Yaskawa INFORM job: R1_W18,19,21(0,0)_KM-OKNEW_MP.JBI

/JOB
//NAME R1_W18,19,21(0,0)_KM-OKNEW_MP
///FOLDERNAME SCIANA-NOWY-R2-KM
//POS
///NPOS 80,80,0,5,0,0
///TOOL 0
///POSTYPE PULSE
///PULSE
C00000=160147,-53341,-73853,12461,99147,-87592
C00001=218993,-28852,-38707,63009,50059,-50724
C00002=220406,-26361,-36985,62252,49273,-50314
C00003=220646,-24565,-35727,62034,49192,-50185
C00004=230254,-40887,-46835,45385,32404,-42165
C00005=230400,-39401,-45908,45036,32465,-41986
C00006=231234,-39623,-46051,44273,32027,-41630
C00007=229297,-43449,-48422,46653,32652,-42787
C00008=220299,-31016,-30594,80800,44642,-56707
C00009=217027,-34239,-32011,82093,46850,-57475
C00010=218993,-28852,-38707,63009,50059,-50724
C00011=218994,-27956,-30243,66729,47934,-53296
C00012=220309,-26407,-29170,66164,47121,-52969
C00013=220627,-24126,-27569,65891,46994,-52801
C00014=226141,-36155,-35714,59251,35589,-49390
C00015=226354,-34126,-34390,58846,35579,-49175
C00016=227436,-34522,-34649,58234,34891,-48867
C00017=226354,-34126,-34390,58846,35579,-49175
C00018=223002,-47340,-42625,62762,36811,-51283
C00019=212788,-54368,-45816,77108,46096,-57028
C00020=192935,-54093,-45665,79683,60227,-58916
C00021=199706,-75247,-47809,90044,85458,-59697
C00022=-183741,-84985,-51911,-73844,36583,24995
C00023=-167288,13673,-10685,-75581,87166,55635
C00024=-170115,12447,-11796,-75038,85255,55349
C00025=-171924,12238,-11987,-74680,84031,55173
C00026=-172522,13420,-10920,-74565,83613,55136
C00027=-171924,12238,-11987,-74680,84031,55173
C00028=-174289,-8390,-27193,-73022,70502,53860
C00029=-175043,-10382,-28758,-72859,69972,53803
C00030=-173781,-9335,-27936,-73156,70837,53929
C00031=-170061,7965,-6237,-85273,82617,57097
C00032=-170115,12447,-11796,-75038,85255,55349
C00033=-170854,10317,-178,-75577,82417,58957
C00034=-171936,11268,672,-75477,81652,58870
C00035=-172588,12571,1843,-75403,81184,58831
C00036=-173506,-7047,-14827,-73481,70592,57186
C00037=-174065,-6013,-13997,-73389,70213,57115
C00038=-174718,-7755,-15385,-73301,69749,57060
C00039=-174065,-6013,-13997,-73389,70213,57115
C00040=-167494,-6216,-14159,-74323,74762,57821
C00041=-167212,9242,-4388,-85630,84611,57426
C00042=-171443,11016,-20134,-69762,86873,53798
C00043=-159366,28260,10505,-84577,79142,62797
C00044=-161376,29134,12959,-84526,77561,63200
C00045=-170734,9630,-20866,-69941,87234,53997
C00046=-170910,12626,-18186,-69900,87078,54023
C00047=-161329,41068,52798,-88533,75848,71873
C00048=-156885,52620,73245,-89064,78615,75095
C00049=-156885,42414,52033,-87693,79106,71429
C00050=-156885,42414,52033,-87693,79106,71429
C00051=-170734,9630,-20866,-69941,87234,53997
C00052=-170910,12626,-18186,-69900,87078,54023
C00053=-157101,42923,53642,-87848,78897,71764
C00054=-152830,31819,8463,-85121,84190,61637
C00055=-158696,27639,4326,-84119,80078,61206
C00056=-161292,29017,11142,-84335,77760,62716
C00057=-170734,9630,-20866,-69941,87234,53997
C00058=-170910,12626,-18186,-69900,87078,54023
C00059=-161298,39658,49489,-88232,75954,71262
C00060=-157285,44272,54296,-87830,78791,71632
C00061=-149677,12279,17067,-86345,84838,68845
C00062=-232880,-71521,-75686,35941,36210,-39067
C00063=-222816,-51916,-50111,20966,8363,-34041
C00064=-221849,-36521,-38911,13718,8860,-30841
C00065=-232908,-27541,-49501,31528,41666,-36518
C00066=-231674,-29527,-50857,30509,41069,-36068
C00067=-221749,-36952,-39190,13316,8793,-30662
C00068=-222742,-43680,-43403,19802,8163,-33549
C00069=-222742,-43680,-43403,19802,8163,-33549
C00070=-222596,-43007,-42997,18855,8220,-33127
C00071=-222188,-38344,-40086,15669,8713,-31707
C00072=-221923,-38189,-39826,14529,8586,-31201
C00073=-222612,-48256,-49120,16792,9247,-32198
C00074=-222612,-48582,-51707,14592,10621,-31204
C00075=-222673,-45322,-48482,15253,10333,-31500
C00076=-222605,-45676,-48694,15053,10272,-31413
C00077=-229461,-68293,-61058,53300,9643,-48481
C00078=-91363,-148629,-70156,-110021,65590,32869
C00079=-795,-65919,-41644,-5435,89623,77465
BC00000=340583,1203205,1070892
BC00001=395849,1203429,1070910
BC00002=395849,1203429,1070910
BC00003=395849,1203429,1070910
BC00004=395849,1203429,1070910
BC00005=395849,1203429,1070910
BC00006=395849,1203429,1070910
BC00007=395849,1203429,1070910
BC00008=395849,1203429,1070910
BC00009=395849,1203429,1070910
BC00010=395849,1203429,1070910
BC00011=395849,1203429,690394
BC00012=395849,1203429,690394
BC00013=395849,1203429,690394
BC00014=395849,1203429,690394
BC00015=395849,1203429,690394
BC00016=395849,1203429,690394
BC00017=395849,1203429,690394
BC00018=395849,1203429,690394
BC00019=395849,1203429,886238
BC00020=395849,1203429,886238
BC00021=392558,1157770,1067511
BC00022=392558,972054,1067511
BC00023=363587,801900,1037584
BC00024=363587,805740,1037584
BC00025=363587,805740,1037584
BC00026=363587,805740,1037584
BC00027=363587,805740,1037584
BC00028=363587,805740,1037584
BC00029=363587,805740,1037584
BC00030=363587,805740,1037584
BC00031=363587,805740,1037584
BC00032=363587,805740,1037584
BC00033=363587,805740,689443
BC00034=363587,805740,689443
BC00035=363586,805740,689440
BC00036=363587,805740,689443
BC00037=363587,805740,689443
BC00038=363587,805740,689443
BC00039=363587,805740,689443
BC00040=363587,805740,689443
BC00041=363587,805740,1037584
BC00042=366059,811819,1070910
BC00043=358283,754245,1070910
BC00044=358283,754245,1070910
BC00045=358283,754245,1070910
BC00046=358283,754245,1070910
BC00047=358283,754245,1070910
BC00048=358283,754245,1069404
BC00049=352744,750822,887513
BC00050=348457,746222,883985
BC00051=358283,754245,1070910
BC00052=358283,754245,1070910
BC00053=348457,746222,705777
BC00054=358284,754245,886289
BC00055=358284,754245,886289
BC00056=358283,754245,886291
BC00057=358283,754245,1070910
BC00058=358283,754245,1070910
BC00059=358283,754245,886291
BC00060=358283,754245,885920
BC00061=358283,794942,867656
BC00062=395849,1135044,1070910
BC00063=395849,1140911,1070910
BC00064=395849,1140998,1070910
BC00065=395849,1142547,1070910
BC00066=395849,1142547,1070910
BC00067=395849,1140998,895189
BC00068=395849,1140998,895189
BC00069=395849,1140998,721535
BC00070=394321,1142791,721535
BC00071=394321,1142791,721535
BC00072=394321,1142791,532615
BC00073=394321,1142791,532615
BC00074=394321,1142791,868876
BC00075=387636,1145223,868873
BC00076=387636,1145223,693943
BC00077=387636,1145223,693943
BC00078=390319,830411,754737
BC00079=219086,754245,1011344
///POSTYPE BASE
///RECTAN
///RCONF 0,0,0,0,0,0,0,0,0,0,0,0,0,0,0,0,0,0,0,0,0,0,0,0
P00006=0.222,-3.123,-1.508,0.0000,0.0000,0.0000
P00026=0.562,-0.002,-0.337,0.0000,0.0000,0.0000
P00027=-0.746,0.015,-9.096,0.0000,0.0000,0.0000
P00028=-2.237,-0.018,-7.702,0.0000,0.0000,0.0000
P00029=-2.156,-0.086,-4.681,0.0000,0.0000,0.0000
//INST
///DATE 2024/07/18 17:23
///ATTR SC,RW
///GROUP1 RB1,BS1
NOP
SFTOF
MOVJ C00000 BC00000 VJ=100.00
MOVL C00001 BC00001 V=500.0
MOVL C00002 BC00002 V=60.0
REFP 3 C00003 BC00003
CALL JOB:SEARCH-R1
SET P027 P006
SFTON P027
MOVL C00004 BC00004 V=60.0
MOVL C00005 BC00005 V=60.0
REFP 3 C00006 BC00006
CALL JOB:SEARCH-R1
SET P027 P006
SFTON P027
MOVL C00007 BC00007 V=60.0
MOVL C00008 BC00008 V=166.7
MOVL C00009 BC00009 V=166.7
'DOL
MOVL C00010 BC00010 V=166.7
MOVL C00011 BC00011 V=166.7
SFTOF
MOVL C00012 BC00012 V=60.0
REFP 3 C00013 BC00013
CALL JOB:SEARCH-R1
SET P029 P006
SFTON P029
MOVL C00014 BC00014 V=60.0
MOVL C00015 BC00015 V=60.0
REFP 3 C00016 BC00016
CALL JOB:SEARCH-R1
SET P029 P006
SFTON P029
MOVL C00017 BC00017 V=60.0
MOVL C00018 BC00018 V=60.0
MOVL C00019 BC00019 V=500.0
MOVL C00020 BC00020 V=500.0
SFTOF
'DRUGA STRONA
MOVJ C00021 BC00021 VJ=40.00
MOVJ C00022 BC00022 VJ=80.00
MOVL C00023 BC00023 V=666.7
MOVL C00024 BC00024 V=333.3
MOVL C00025 BC00025 V=83.3
REFP 3 C00026 BC00026
CALL JOB:SEARCH-R1
SET P026 P006
SFTON P026
MOVL C00027 BC00027 V=100.0
MOVL C00028 BC00028 V=100.0
REFP 3 C00029 BC00029
CALL JOB:SEARCH-R1
SET P026 P006
SFTON P026
MOVL C00030 BC00030 V=166.7
SFTOF
MOVL C00031 BC00031 V=333.3
'DOL
MOVL C00032 BC00032 V=166.7
MOVL C00033 BC00033 V=166.7
MOVL C00034 BC00034 V=60.0
REFP 3 C00035 BC00035
CALL JOB:SEARCH-R1
SET P028 P006
SFTON P028
MOVL C00036 BC00036 V=60.0
MOVL C00037 BC00037 V=60.0
REFP 3 C00038 BC00038
CALL JOB:SEARCH-R1
SET P028 P006
SFTON P028
MOVL C00039 BC00039 V=60.0
MOVL C00040 BC00040 V=333.3
MOVL C00041 BC00041 V=500.0
'Path S879 (for W18)
SFTOF
SFTON P026
MOVL C00042 BC00042 V=500.0
MOVL C00043 BC00043 V=333.3
MOVL C00044 BC00044 V=166.7 PL=0
REFP 1 C00045 BC00045
REFP 2 C00046 BC00046
MACRO1 MJ#(0) ARGF6
ARCON
MOVL C00047 BC00047 V=13.3
ARCOF
'Path W883_C
SFTOF
SFTON P028
MOVL C00048 BC00048 V=250.0
MOVL C00049 BC00049 V=333.3
MOVL C00050 BC00050 V=100.0 PL=0
REFP 1 C00051 BC00051
REFP 2 C00052 BC00052
MACRO1 MJ#(0) ARGF6
ARCON
MOVL C00053 BC00053 V=13.3
ARCOF
'Path W883_B
SFTOF
SFTON P028
MOVL C00054 BC00054 V=333.3
MOVL C00055 BC00055 V=333.3
MOVL C00056 BC00056 V=166.7 PL=0
REFP 1 C00057 BC00057
REFP 2 C00058 BC00058
MACRO1 MJ#(0) ARGF6
ARCON
SFTON P028
MOVL C00059 BC00059 V=13.3
ARCOF
MOVL C00060 BC00060 V=250.0
SFTOF
MOVL C00061 BC00061 V=333.3
MOVL C00062 BC00062 V=333.3
MOVL C00063 BC00063 V=166.7
SFTON P027
MOVL C00064 BC00064 V=166.7 PL=0
REFP 1 C00065 BC00065
REFP 2 C00066 BC00066
MACRO1 MJ#(0) ARGF6
ARCON
MOVL C00067 BC00067 V=12.5
ARCOF
MOVL C00068 BC00068 V=166.7
SFTOF
MOVJ C00069 BC00069 VJ=100.00
SFTON P029
MOVJ C00070 BC00070 VJ=100.00
MACRO1 MJ#(0) ARGF6
MOVL C00071 BC00071 V=116.7 PL=0
ARCON
MOVL C00072 BC00072 V=12.5
ARCOF
TIMER T=1.00
SFTOF
MOVJ C00073 BC00073 VJ=100.00
MOVJ C00074 BC00074 VJ=50.00
SFTON P029
MOVJ C00075 BC00075 VJ=20.00 PL=0
ARCON
MOVL C00076 BC00076 V=12.5
ARCOF
TIMER T=1.00
SFTOF
MOVL C00077 BC00077 V=333.3
SFTOF
MOVJ C00078 BC00078 VJ=100.00
MOVJ C00079 BC00079 VJ=100.00
END
